Fanuc KAREL source: KCL_STATUS.kl

PROGRAM T
%NOLOCKGROUP
VAR
 res : INTEGER
BEGIN
 res = KCL_STATUS
END T
